// TIA Portal V20 export
TYPE "type_emRelations_em2_SoftCam"
// stored: Access Published, Namespace Unit1
   STRUCT
      jrOutPnPLeftAxisX : Struct
         pos00_wait : "LER_typeSoftCamPosition";
         pos01_stack1Load : "LER_typeSoftCamPosition";
         pos02_stack2Load : "LER_typeSoftCamPosition";
         pos03_unload : "LER_typeSoftCamPosition";
         pos04_posistion { ExternalWritable := 'False'} : "LER_typeSoftCamPosition";
         pos05_posistion { ExternalWritable := 'False'} : "LER_typeSoftCamPosition";
         pos06_posistion { ExternalWritable := 'False'} : "LER_typeSoftCamPosition";
         pos07_posistion { ExternalWritable := 'False'} : "LER_typeSoftCamPosition";
         pos08_noInterferenceZone { ExternalWritable := 'False'} : "LER_typeSoftCamPosition";
         pos09_stack1LoadZone : "LER_typeSoftCamPosition";
         pos10_stack2LoadZone : "LER_typeSoftCamPosition";
         pos11_unloadZone : "LER_typeSoftCamPosition";
         pos12_posistion : "LER_typeSoftCamPosition";
         pos13_posistion { ExternalWritable := 'False'} : "LER_typeSoftCamPosition";
         pos14_posistion { ExternalWritable := 'False'} : "LER_typeSoftCamPosition";
         pos15_posistion { ExternalWritable := 'False'} : "LER_typeSoftCamPosition";
      END_STRUCT;
      jrOutPnPLeftAxisZ : Struct
         pos00_wait : "LER_typeSoftCamPosition";
         pos01_stack1Load : "LER_typeSoftCamPosition";
         pos02_stack2Load : "LER_typeSoftCamPosition";
         pos03_unload : "LER_typeSoftCamPosition";
         pos04_posistion { ExternalWritable := 'False'} : "LER_typeSoftCamPosition";
         pos05_posistion { ExternalWritable := 'False'} : "LER_typeSoftCamPosition";
         pos06_posistion { ExternalWritable := 'False'} : "LER_typeSoftCamPosition";
         pos07_posistion { ExternalWritable := 'False'} : "LER_typeSoftCamPosition";
         pos08_noInterferenceZone { ExternalWritable := 'False'} : "LER_typeSoftCamPosition";
         pos09_posistion : "LER_typeSoftCamPosition";
         pos10_posistion { ExternalWritable := 'False'} : "LER_typeSoftCamPosition";
         pos11_posistion { ExternalWritable := 'False'} : "LER_typeSoftCamPosition";
         pos12_posistion { ExternalWritable := 'False'} : "LER_typeSoftCamPosition";
         pos13_posistion { ExternalWritable := 'False'} : "LER_typeSoftCamPosition";
         pos14_posistion { ExternalWritable := 'False'} : "LER_typeSoftCamPosition";
         pos15_posistion { ExternalWritable := 'False'} : "LER_typeSoftCamPosition";
      END_STRUCT;
      jrOutPnPRightAxisX : Struct
         pos00_wait : "LER_typeSoftCamPosition";
         pos01_load : "LER_typeSoftCamPosition";
         pos02_unload : "LER_typeSoftCamPosition";
         pos03_posistion { ExternalWritable := 'False'} : "LER_typeSoftCamPosition";
         pos04_posistion { ExternalWritable := 'False'} : "LER_typeSoftCamPosition";
         pos05_posistion { ExternalWritable := 'False'} : "LER_typeSoftCamPosition";
         pos06_posistion { ExternalWritable := 'False'} : "LER_typeSoftCamPosition";
         pos07_posistion { ExternalWritable := 'False'} : "LER_typeSoftCamPosition";
         pos08_noInterferenceZone { ExternalWritable := 'False'} : "LER_typeSoftCamPosition";
         pos09_loadZone : "LER_typeSoftCamPosition";
         pos10_unloadZone : "LER_typeSoftCamPosition";
         pos11_posistion : "LER_typeSoftCamPosition";
         pos12_posistion { ExternalWritable := 'False'} : "LER_typeSoftCamPosition";
         pos13_posistion { ExternalWritable := 'False'} : "LER_typeSoftCamPosition";
         pos14_posistion { ExternalWritable := 'False'} : "LER_typeSoftCamPosition";
         pos15_posistion { ExternalWritable := 'False'} : "LER_typeSoftCamPosition";
      END_STRUCT;
      jrOutPnPRightAxisZ : Struct
         pos00_wait : "LER_typeSoftCamPosition";
         pos01_load : "LER_typeSoftCamPosition";
         pos02_unload : "LER_typeSoftCamPosition";
         pos03_posistion { ExternalWritable := 'False'} : "LER_typeSoftCamPosition";
         pos04_posistion { ExternalWritable := 'False'} : "LER_typeSoftCamPosition";
         pos05_posistion { ExternalWritable := 'False'} : "LER_typeSoftCamPosition";
         pos06_posistion { ExternalWritable := 'False'} : "LER_typeSoftCamPosition";
         pos07_posistion { ExternalWritable := 'False'} : "LER_typeSoftCamPosition";
         pos08_noInterferenceZone { ExternalWritable := 'False'} : "LER_typeSoftCamPosition";
         pos09_position : "LER_typeSoftCamPosition";
         pos10_posistion { ExternalWritable := 'False'} : "LER_typeSoftCamPosition";
         pos11_posistion { ExternalWritable := 'False'} : "LER_typeSoftCamPosition";
         pos12_posistion { ExternalWritable := 'False'} : "LER_typeSoftCamPosition";
         pos13_posistion { ExternalWritable := 'False'} : "LER_typeSoftCamPosition";
         pos14_posistion { ExternalWritable := 'False'} : "LER_typeSoftCamPosition";
         pos15_posistion { ExternalWritable := 'False'} : "LER_typeSoftCamPosition";
      END_STRUCT;
   END_STRUCT;
END_TYPE
